// TIA Portal V21 export
TYPE "Std_DatiGetPut"
   STRUCT
      PUT : Struct
         REQ : Bool;   // Trigger Command
         DONE : Bool;   // Data Done
         ERROR : Bool;   // Error Active
         ERROR_PULSE : Bool;   // Error Active
         x04 : Bool;
         x05 : Bool;
         x06 : Bool;
         ALLARM : Bool;   // Comunication Allarm
         ID : Word;   // Channel Number
         i04 : Int;
         w06 : Word;
         w08 : Word;
         STATUS : Word;   // Status
         ATTEMPTS : Int;   // Comunication Attempts
         STATUS_ARRAY_01 : Word;   // Status Store 01
         STATUS_ARRAY_02 : Word;   // Status Store 02
         STATUS_ARRAY_03 : Word;   // Status Store 03
      END_STRUCT;
      GET : Struct
         REQ : Bool;   // Trigger Command
         NDR : Bool;   // Data Done
         ERROR : Bool;   // Error Active
         ERROR_PULSE : Bool;   // Error Active
         x04 : Bool;
         x05 : Bool;
         x06 : Bool;
         ALLARM : Bool;   // Comunication Allarm
         ID : Word;   // Channel Number
         i04 : Int;
         i06 : Int;
         STATUS : Word;   // Status
         w10 : Word;
         ATTEMPTS : Int;   // Comunication Attempts
         STATUS_ARRAY_01 : Word;   // Status Store 01
         STATUS_ARRAY_02 : Word;   // Status Store 02
         STATUS_ARRAY_03 : Word;   // Status Store 03
      END_STRUCT;
   END_STRUCT;
END_TYPE
